{attribute 'GeneratedUsingTerminal: EL6001-0000-0020'}
{attribute addProperty BoxType "EL6001-0000-0020"}
{attribute addProperty Id "AdsAddrAT %I*AMSADDR8StateAT %I*UINT2"}
{attribute addProperty CRC "854291690"}
{attribute addProperty Size "10"}
TYPE InfoData_32EB74EA :
STRUCT
	{attribute addProperty Name "AdsAddr"}
	AdsAddr AT %I* : AMSADDR;
	{attribute addProperty Name "State"}
	State AT %I* : UINT;
END_STRUCT
END_TYPE

(* stored: Version 1.2.0.0, ProductVersion 3.1.4024.9
   DUT InfoData_32EB74EA: Id {f800b426-9c41-4daa-a6e0-ce36f8a11be1} *)
